// Mitsubishi GX Works2 project: test   PLC: Q02U

PROGRAM MAIN
VAR
  test_1 : test;
END_VAR
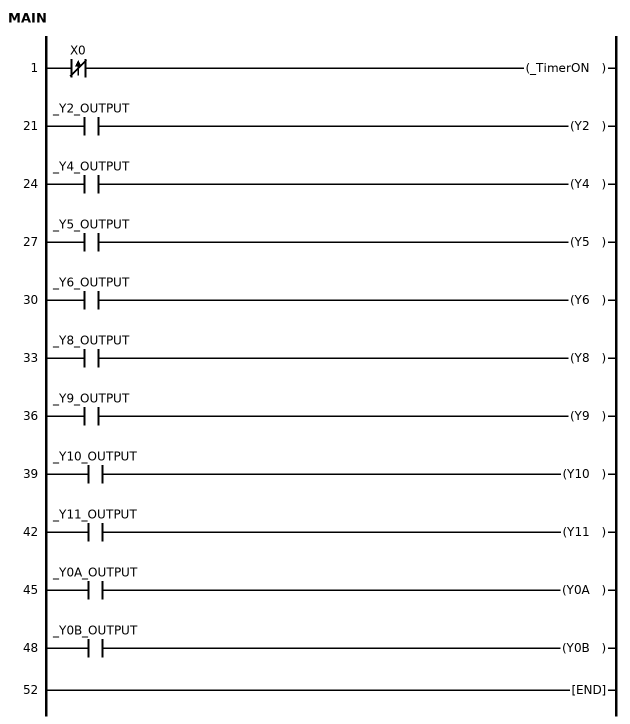
; FB BLK START test(test_1)
1     LDPI    X0
      OUT     _TimerON
; FB START
; FB_NAME test
; INSTANCE_NAME test_1
; FB IN_B:TimerON
; FB OUT_Y2_OUTPUT:B
; FB OUT_Y4_OUTPUT:B
; FB OUT_Y5_OUTPUT:B
; FB OUT_Y6_OUTPUT:B
; FB OUT_Y8_OUTPUT:B
; FB OUT_Y9_OUTPUT:B
; FB OUT_Y10_OUTPUT:B
; FB OUT_Y11_OUTPUT:B
; FB OUT_Y0A_OUTPUT:B
; FB OUT_Y0B_OUTPUT:B
; FB END
21    LD      _Y2_OUTPUT
      OUT     Y2
24    LD      _Y4_OUTPUT
      OUT     Y4
27    LD      _Y5_OUTPUT
      OUT     Y5
30    LD      _Y6_OUTPUT
      OUT     Y6
33    LD      _Y8_OUTPUT
      OUT     Y8
36    LD      _Y9_OUTPUT
      OUT     Y9
39    LD      _Y10_OUTPUT
      OUT     Y10
42    LD      _Y11_OUTPUT
      OUT     Y11
45    LD      _Y0A_OUTPUT
      OUT     Y0A
48    LD      _Y0B_OUTPUT
      OUT     Y0B
; FB BLK END
52    END
END_PROGRAM

FUNCTION_BLOCK test
VAR_INPUT
  TimerON : BOOL;
END_VAR
VAR_OUTPUT
  Y4_OUTPUT : BOOL;
  Y5_OUTPUT : BOOL;
  Y6_OUTPUT : BOOL;
  Y8_OUTPUT : BOOL;
  Y9_OUTPUT : BOOL;
  Y10_OUTPUT : BOOL;
  Y11_OUTPUT : BOOL;
  Y0A_OUTPUT : BOOL;
  Y0B_OUTPUT : BOOL;
  Y2_OUTPUT : BOOL;
END_VAR
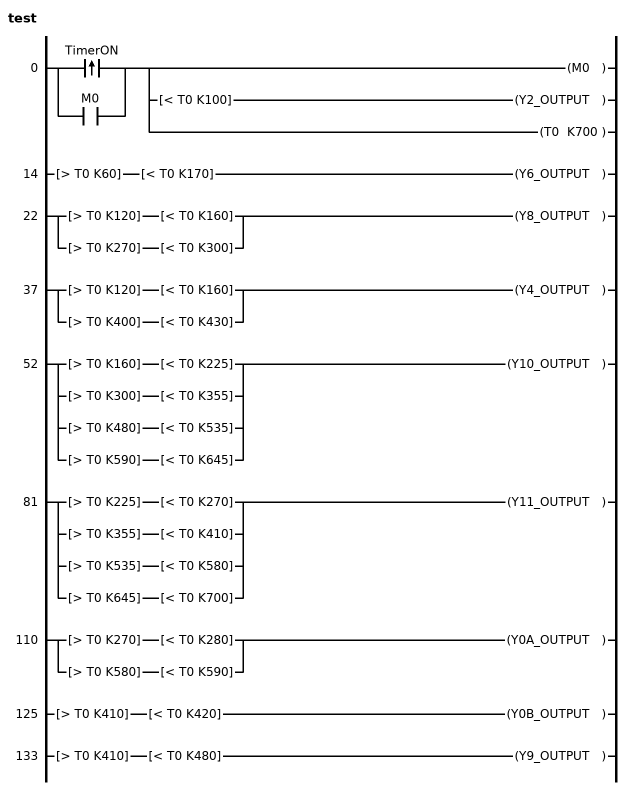
0     LDP     TimerON
      OR      M0
      OUT     M0
      MPS
      AND<    T0 K100
      OUT     Y2_OUTPUT
      MPP
      OUT     T0 K700
14    LD>     T0 K60
      AND<    T0 K170
      OUT     Y6_OUTPUT
22    LD>     T0 K120
      AND<    T0 K160
      LD>     T0 K270
      AND<    T0 K300
      ORB
      OUT     Y8_OUTPUT
37    LD>     T0 K120
      AND<    T0 K160
      LD>     T0 K400
      AND<    T0 K430
      ORB
      OUT     Y4_OUTPUT
52    LD>     T0 K160
      AND<    T0 K225
      LD>     T0 K300
      AND<    T0 K355
      ORB
      LD>     T0 K480
      AND<    T0 K535
      ORB
      LD>     T0 K590
      AND<    T0 K645
      ORB
      OUT     Y10_OUTPUT
81    LD>     T0 K225
      AND<    T0 K270
      LD>     T0 K355
      AND<    T0 K410
      ORB
      LD>     T0 K535
      AND<    T0 K580
      ORB
      LD>     T0 K645
      AND<    T0 K700
      ORB
      OUT     Y11_OUTPUT
110   LD>     T0 K270
      AND<    T0 K280
      LD>     T0 K580
      AND<    T0 K590
      ORB
      OUT     Y0A_OUTPUT
125   LD>     T0 K410
      AND<    T0 K420
      OUT     Y0B_OUTPUT
133   LD>     T0 K410
      AND<    T0 K480
      OUT     Y9_OUTPUT
END_FUNCTION_BLOCK
